PROGRAM MAIN

VAR
	//S1 : digitalInputSensor;
	temp_S : BOOL;
	digitalInputSensor: INT;
	materialTrayInstallationSensor: INT;
END_VAR

//S1();
//S1(on := IOs.S1, inTime := T#50MS, digitalFiltered => temp_S);

//digitalInputSensor.materialTrayInstallationSensor(temp_S);

END_PROGRAM

(* stored: Version 1.1.0.1, ProductVersion 3.1.4024.14
   POU MAIN: Id {71b4f007-c74f-4713-8031-06c83cc6195e}, SpecialFunc None *)
